// TIA Portal V21 export
FUNCTION "SimpleDevice" : Void   // FC580, LAD
{ S7_Optimized_Access := 'TRUE' }
// stored: AutoNumber false, SetENOAutomatically false
   VAR_INPUT
      FI_START : Bool;
      FI_SERVICE : Bool;
   END_VAR
   VAR_OUTPUT
      FQ_OUTPUT : Bool;
   END_VAR
   VAR_IN_OUT
      FIQ_MANUAL : Bool;
      FIQ_Icon : Int;
   END_VAR
   VAR_TEMP
      tempOut : Bool;
   END_VAR
BEGIN

REGION Network 1: OUTPUT
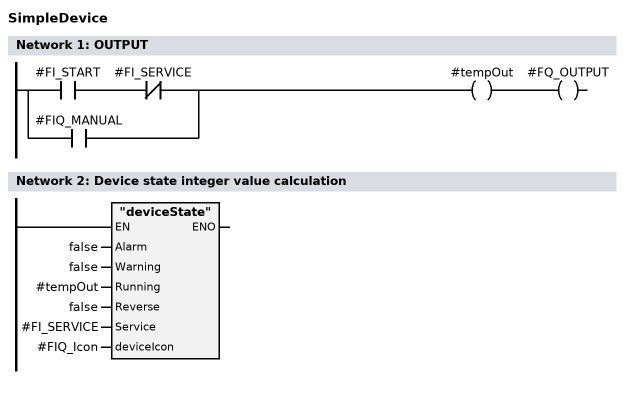
   RUNG wire#powerrail
      Contact( #FI_START )
      I_Contact( #FI_SERVICE )
      wire#w1
      Coil( #tempOut )
      Coil( #FQ_OUTPUT )
   END_RUNG
   RUNG wire#powerrail
      Contact( #FIQ_MANUAL )
   END_RUNG wire#w1
   // the same network as SCL:
   #tempOut := (#FI_START AND NOT #FI_SERVICE) OR #FIQ_MANUAL;
   #FQ_OUTPUT := #tempOut;
END_REGION

REGION Network 2: Device state integer value calculation
   RUNG wire#powerrail
      "deviceState"(Alarm := false, Warning := false, Running := #tempOut, Reverse := false, Service := #FI_SERVICE, deviceIcon := #FIQ_Icon)
   END_RUNG
   // the same network as SCL:
   "deviceState"(Alarm := false,
                 Warning := false,
                 Running := #tempOut,
                 Reverse := false,
                 Service := #FI_SERVICE,
                 deviceIcon := #FIQ_Icon);
END_REGION
END_FUNCTION
